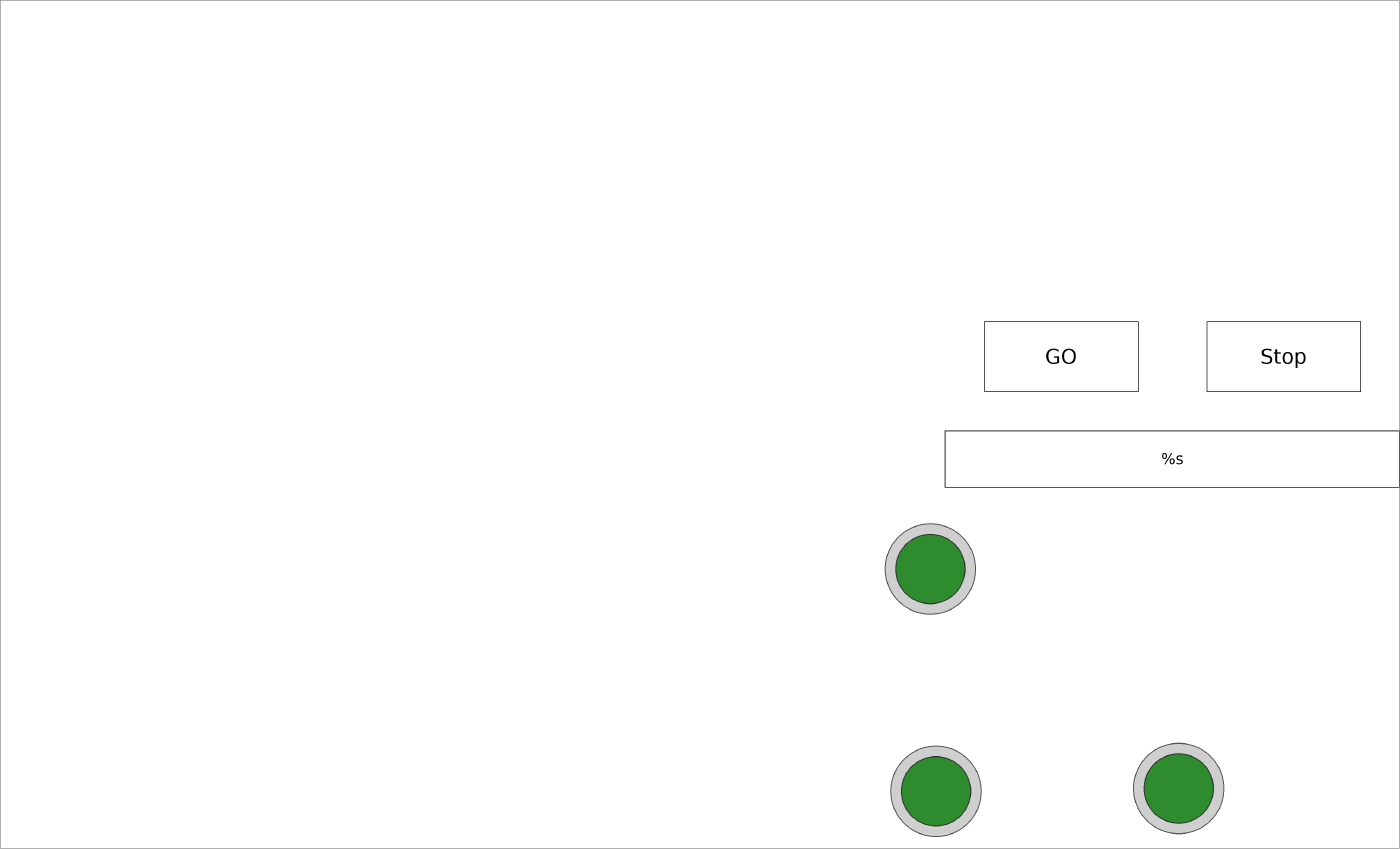
VISUALIZATION Visualization  // 1990x1207
    Lamp1 (1247,727 151x164), variable: GVL.oMainContactor, style: Lamp-Lamp1-Green
    Lamp1 (1600,1039 151x164), variable: GVL.oStarContactor, style: Lamp-Lamp1-Green
    Lamp1 (1255,1043 151x164), variable: GVL.oDeltaContactor, style: Lamp-Lamp1-Green
    Rectangle (1399,457 219x100), "GO"
        OnMouseDown: execute { GVL.iStartPB := true; }
        OnMouseUp: execute { GVL.iStartPB := false; }
    Rectangle (1715,457 219x100), "Stop"
        OnMouseDown: execute { GVL.iStopPB := true; }
        OnMouseUp: execute { GVL.iStopPB := false; }
    Rectangle (1343,612 647x81), "%s", text variable: GVL.oState
END_VISUALIZATION

(* stored: Version 1.1.0.1, ProductVersion 3.1.4024.10
   Visu Visualization: Id {1e6f0995-b575-4d32-9928-96b93441be22} *)
